(* IEC 61131-3 sources: sigmatek-logger-api/IXON_API/Class/IXON_LoggerAPI_Interface, 1 file *)

(* ---- IXON_LoggerAPI_Interface.st ---- *)
#define SND_DATA_ARRAY_SIZE 1024
#define SND_ARRAY_SIZE 20
#define RCV_DATA_ARRAY_SIZE 1024

(*!
<Class
	Name               = "IXON_LoggerAPI_Interface"
	Revision           = "0.0"
	RealtimeTask       = "false"
	CyclicTask         = "true"
	DefCyclictime      = "10 ms"
	BackgroundTask     = "false"
	Sigmatek           = "false"
	OSInterface        = "false"
	HighPriority       = "false"
	Automatic          = "false"
	UpdateMode         = "Prescan"
	SharedCommandTable = "true"
	Objectsize         = "(810,360)">
	<Channels>
		<Server Name="sIPAddrIXON" Class="String" Visualized="true" Remotely="true" Initialize="true" WriteProtected="false" Retentive="false" Comment="use this channel to access the string functions"/>
		<Server Name="sIPAddrPLC" Class="String" Visualized="true" Remotely="true" Initialize="true" WriteProtected="false" Retentive="false" Comment="use this channel to access the string functions"/>
		<Server Name="sPasswordIXON" Class="String" Visualized="true" Remotely="true" Initialize="true" WriteProtected="false" Retentive="false" Comment="use this channel to access the string functions"/>
		<Server Name="sRcvCnt" Visualized="false" Initialize="false" WriteProtected="true" Retentive="false"/>
		<Server Name="sReconnectDelay" Visualized="true" Remotely="true" Initialize="true" DefValue="10000" WriteProtected="false" Retentive="false"/>
		<Server Name="sSendDelay" Visualized="true" Remotely="true" Initialize="true" DefValue="200" WriteProtected="false" Retentive="false"/>
		<Server Name="sSndCnt" Visualized="false" Initialize="false" WriteProtected="true" Retentive="false"/>
		<Server Name="sTCPStep" Visualized="true" Remotely="true" Initialize="false" WriteProtected="false" Retentive="false"/>
		<Client Name="_StdLib" Required="false" Internal="false"/>
		<Client Name="ST_IPAddrIXON" Required="true" Internal="true"/>
		<Client Name="ST_IPAddrPLC" Required="true" Internal="true"/>
		<Client Name="ST_PasswordIXON" Required="true" Internal="true"/>
	</Channels>
	<Separators>
		<Servers>
			<SepChn Position="0"/>
			<SepChn Position="6"/>
		</Servers>
	</Separators>
	<Network Name="IXON_LoggerAPI_Interface">
		<!-- List of Components in this network -->
		<Components>
			<Object
				Name       = "_base"
				Class      = "_TCPIPClientInterface"
				Position   = "(218,120)"
				Visualized = "false">
				<Channels>
					<Server Name="ClassSvr"/>
					<Server Name="ErrorCode"/>
					<Server Name="ErrorGroup"/>
					<Server Name="ErrorState"/>
					<Server Name="State"/>
					<Client Name="_TCPIPClient"/>
				</Channels>
			</Object>
			<Object
				Name       = "ST_IPAddrIXON"
				Class      = "String"
				Position   = "(210,510)"
				Visualized = "true"
				Remotely   = "true">
				<Channels>
					<Server Name="Data"/>
					<Client Name="SingleRealloc" Value="1"/>
				</Channels>
			</Object>
			<Object
				Name       = "ST_IPAddrPLC"
				Class      = "String"
				Position   = "(210,660)"
				Visualized = "true"
				Remotely   = "true">
				<Channels>
					<Server Name="Data"/>
					<Client Name="SingleRealloc" Value="1"/>
				</Channels>
			</Object>
			<Object
				Name       = "ST_PasswordIXON"
				Class      = "String"
				Position   = "(210,810)"
				Visualized = "true"
				Remotely   = "true">
				<Channels>
					<Server Name="Data"/>
					<Client Name="SingleRealloc" Value="1"/>
				</Channels>
			</Object>
		</Components>
		<Comments>
		</Comments>
		<!-- List of Connections in this network -->
		<Connections>
			<Connection Source="this.ClassSvr" Destination="_base.ClassSvr" Vertices="(1096,210),(924,210),"/>
			<Connection Source="this.State" Destination="_base.State" Vertices="(1096,270),(924,270),"/>
			<Connection Source="this.ErrorState" Destination="_base.ErrorState" Vertices="(1096,330),(924,330),"/>
			<Connection Source="this.ErrorGroup" Destination="_base.ErrorGroup" Vertices="(1096,390),(924,390),"/>
			<Connection Source="this.ErrorCode" Destination="_base.ErrorCode" Vertices="(1096,450),(924,450),"/>
			<Connection Source="_base._TCPIPClient" Destination="this._TCPIPClient" Vertices="(218,210),(38,210),"/>
			<Connection Source="this.ST_IPAddrIXON" Destination="ST_IPAddrIXON.Data"/>
			<Connection Source="this.sIPAddrIXON" Destination="ST_IPAddrIXON.Data" Vertices="(1096,510),(586,600),"/>
			<Connection Source="this.ST_PasswordIXON" Destination="ST_PasswordIXON.Data"/>
			<Connection Source="this.sPasswordIXON" Destination="ST_PasswordIXON.Data" Vertices="(1096,630),(586,900),"/>
			<Connection Source="this.ST_IPAddrPLC" Destination="ST_IPAddrPLC.Data"/>
			<Connection Source="this.sIPAddrPLC" Destination="ST_IPAddrPLC.Data" Vertices="(1096,570),(586,750),"/>
		</Connections>
		<!-- Headerfiles -->
		<Options>
		</Options>
	</Network>
</Class>
*)
#pragma using _TCPIPClientInterface

IXON_LoggerAPI_Interface : CLASS
: _TCPIPClientInterface
	TYPE
	  teUSER_TCP_STEPS :  //! <Type Public="true" Name="teUSER_TCP_STEPS"/>
	  (
	    UTS_Idle,
	    UTS_Connect,
	    UTS_CheckConnect,
	    UTS_ConnectIXON,
	    UTS_WaitConnectIXON,
	    UTS_WaitData,
	    UTS_SendData,
	    UTS_WaitSendData,
	    UTS_Disconnect,
	    UTS_Error
	  )$UDINT;
	END_TYPE
  //Servers:
	sIPAddrIXON 	: SvrChCmd_UDINT;
	sIPAddrPLC 	: SvrChCmd_UDINT;
	sPasswordIXON 	: SvrChCmd_UDINT;
	sSendDelay 	: SvrCh_UDINT;
	sReconnectDelay 	: SvrCh_UDINT;
	sTCPStep 	: SvrCh_teUSER_TCP_STEPS_PTofCls_IXON_LoggerAPI_Interface;
	sSndCnt 	: SvrCh_DINT;
	sRcvCnt 	: SvrCh_DINT;
  //Clients:
	_StdLib 	: CltChCmd__StdLib;
	ST_IPAddrIXON 	: CltChCmd_String;
	ST_PasswordIXON 	: CltChCmd_String;
	ST_IPAddrPLC 	: CltChCmd_String;
  //Variables:
		vSendData : ARRAY [0..SND_ARRAY_SIZE-1, 0..SND_DATA_ARRAY_SIZE-1] OF CHAR;

		vSendDataIndex 	: DINT;
		vRcvData : ARRAY [0..RCV_DATA_ARRAY_SIZE-1] OF CHAR;

		vRcvNewData 	: DINT;
		vLength 	: UDINT;
		vLocIPAddress : ARRAY [0..15] OF CHAR;

		vIsConnected 	: BOOL;
		vTcpTimeOut 	: UDINT;
		vCheckConnectionIXON 	: UDINT;
		vTimeMark 	: UDINT;
		VTimeMark2 	: UDINT;
		vIntError 	: DINT;
		vConnectData : ARRAY [0..100] OF CHAR;

		vSendRepeat 	: DINT;
  //Functions:

	FUNCTION VIRTUAL GLOBAL Init;

	FUNCTION VIRTUAL GLOBAL CyWork
		VAR_INPUT
			EAX 	: UDINT;
		END_VAR
		VAR_OUTPUT
			state (EAX) 	: UDINT;
		END_VAR;
				//! <Function Comment="This Method is called if Data is received (Overwrite it)&#13;&#10;For receiving a spezial amount of Data you have to use the &#13;&#10;DataHandling Methode." Name="Response"/>
	FUNCTION VIRTUAL GLOBAL Response
		VAR_INPUT
			pData 	: ^void;			//! <Variable Comment="Pointer to Data" Name="Response.pData"/>
			udsize 	: UDINT;			//! <Variable Comment="Size of Data" Name="Response.udsize"/>
		END_VAR;

	FUNCTION GLOBAL AddStringToBuffer
		VAR_INPUT
			pData 	: ^void;
			udLen 	: UDINT;
		END_VAR;

	FUNCTION VIRTUAL GLOBAL sIPAddrIXON::Read
		VAR_OUTPUT
			output (EAX) 	: UDINT;
		END_VAR;

	FUNCTION VIRTUAL GLOBAL sIPAddrIXON::Write
		VAR_INPUT
			input (EAX) 	: UDINT;
		END_VAR
		VAR_OUTPUT
			result (EAX) 	: UDINT;
		END_VAR;

	FUNCTION VIRTUAL GLOBAL sIPAddrPLC::Read
		VAR_OUTPUT
			output (EAX) 	: UDINT;
		END_VAR;

	FUNCTION VIRTUAL GLOBAL sIPAddrPLC::Write
		VAR_INPUT
			input (EAX) 	: UDINT;
		END_VAR
		VAR_OUTPUT
			result (EAX) 	: UDINT;
		END_VAR;

	FUNCTION VIRTUAL GLOBAL sPasswordIXON::Read
		VAR_OUTPUT
			output (EAX) 	: UDINT;
		END_VAR;

	FUNCTION VIRTUAL GLOBAL sPasswordIXON::Write
		VAR_INPUT
			input (EAX) 	: UDINT;
		END_VAR
		VAR_OUTPUT
			result (EAX) 	: UDINT;
		END_VAR;
  //Tables:
	FUNCTION @STD
		VAR_OUTPUT
			ret_code	: CONFSTATES;
		END_VAR;
	FUNCTION GLOBAL TAB @CT_;
END_CLASS;

#pragma using String
#pragma usingLtd _StdLib

FUNCTION VIRTUAL GLOBAL IXON_LoggerAPI_Interface::Init
  VAR
  	index : UDINT;
  END_VAR

  if _FirstScan then
    vTcpTimeOut := 2000 ms;
    vCheckConnectionIXON := 10000 ms;
    vTimeMark := ops.tAbsolute := 10000 ms;
  end_if;
END_FUNCTION

FUNCTION VIRTUAL GLOBAL IXON_LoggerAPI_Interface::CyWork
	VAR_INPUT
		EAX 	: UDINT;
	END_VAR
	VAR_OUTPUT
		state (EAX) 	: UDINT;
	END_VAR
  VAR
  	retCode : DINT;
    index : UDINT;
    length : UDINT;
    i : INT;
  END_VAR

  // ==========================================================================
  case sTCPStep of

    // --------------------------------------------------------------
    UTS_Idle:
      if (ops.tAbsolute - vTimeMark) > 1000 ms then
        sTCPStep := UTS_Connect;
      end_if;

    // --------------------------------------------------------------
    UTS_Connect:

      vLength := ST_IPAddrIXON.GetLength();

      if vLength > sizeof(vLocIPAddress) then
        vTimeMark := ops.tAbsolute;
        vIntError := -1; // IP address too long.
        sTCPStep := UTS_Error;
        return;
      end_if;

      ST_IPAddrIXON.GetDataAt(pData:=#vLocIPAddress[0],
                                 udSize:=vLength,
                                 udAt:=0);

      vLocIPAddress[vLength]:=0;

      retCode := AddConnection(pIPAddress:=#vLocIPAddress[0],
                               udTimeout:= 0);

      if retCode > 0 then
        vTimeMark := ops.tAbsolute;
        sTCPStep := UTS_CheckConnect;
      else
        vTimeMark := ops.tAbsolute;
        vIntError := -2; // Connection could not be established.
        sTCPStep := UTS_Error;
        return;
      end_if;

    // --------------------------------------------------------------
    UTS_CheckConnect:

      if vRcvNewData = 1 then
        vRcvNewData := 0;
        if _memcmp(ptr1:=#vRcvData[0], ptr2:="HELO", cntr:=4) = 0 then
          sTCPStep := UTS_ConnectIXON;
        end_if;
      end_if;
      if (ops.tAbsolute - vTimeMark) > vTcpTimeOut  then
        sTCPStep := UTS_Disconnect;
      end_if;

    // --------------------------------------------------------------
    UTS_ConnectIXON:

      _strcpy(dest:=#vConnectData[0], src:="DEVC ");
      length := ST_IPAddrPLC.GetLength();
      ST_IPAddrPLC.GetDataAt(pData:=#vConnectData[5], udSize:=length, udAt:=0);
      index := 5 + length;
      _strcat(dest:=#vConnectData[index], src:=" ");
      length := ST_PasswordIXON.GetLength();
      index := index + 1;
      ST_PasswordIXON.GetDataAt(pData:=#vConnectData[index], udSize:=length, udAt:=0);
      index := index + length;
      vConnectData[index] := 16#0a;
      vConnectData[index + 1] := 0;

      retCode := SendData(pData:=#vConnectData[0],
                          udSize:= index + 1,
                          bDirect:=TRUE);

      if retCode = 0 then
        vTimeMark := ops.tAbsolute;
        sTCPStep := UTS_WaitConnectIXON;
      else
        vTimeMark := ops.tAbsolute;
        vIntError := -11; // Error connecting IXON
        sTCPStep := UTS_Error;
        return;
      end_if;

    // --------------------------------------------------------------
    UTS_WaitConnectIXON:

      if vRcvNewData = 1 then
        vRcvNewData := 0;
        if _memcmp(ptr1:=#vRcvData[0], ptr2:="DEVC OK", cntr:=7) = 0 then
          vTimeMark := ops.tAbsolute;
          sTCPStep := UTS_WaitData;
        end_if;
      end_if;
      if (ops.tAbsolute - vTimeMark) > vTcpTimeOut  then
        vIntError := -12; // Error connecting IXON response
        sTCPStep := UTS_Error;
      end_if;

    // --------------------------------------------------------------
    UTS_WaitData:

      vIsConnected := IsConnected();

      if vIsConnected = FALSE then
        sTCPStep := UTS_Disconnect;
      elsif _strlen(src:=#vSendData[0][0]) > 0 & (ops.tAbsolute - VTimeMark2) > sSendDelay then
        sTCPStep := UTS_SendData;
      elsif (ops.tAbsolute - vTimeMark) > vCheckConnectionIXON  then
        sTCPStep := UTS_ConnectIXON;
      end_if;

    // --------------------------------------------------------------
    UTS_SendData:

      retCode := SendData(pData:=#vSendData[0][0],
                          udSize:= _strlen(src:=#vSendData[0][0]),
                          bDirect:=TRUE);

      if retCode = 0 then
        for i := 0 to SND_ARRAY_SIZE - 2 do
          vSendData[i] := vSendData[i + 1];
        end_for;
        _strcpy(dest:=#vSendData[SND_ARRAY_SIZE - 1][0], src:="");
        vSendDataIndex -= 1;

        sSndCnt += 1;
        vTimeMark := ops.tAbsolute;
        vTimeMark2 := ops.tAbsolute;
        vSendRepeat := 0;
        sTCPStep := UTS_WaitData; //UTS_WaitSendData;
      else
        vTimeMark := ops.tAbsolute;
        vIntError := -3; // Error sending data
        sTCPStep := UTS_Error;
        return;
      end_if;

    // --------------------------------------------------------------
    UTS_WaitSendData:

      if (ops.tAbsolute - vTimeMark) > vTcpTimeOut  then
        sTCPStep := UTS_Disconnect;
      end_if;

    // --------------------------------------------------------------
    UTS_Disconnect:

      retCode := DelConnection();

      if retCode  = TCP_CLT_NO_ERROR then
        vTimeMark := ops.tAbsolute;
        sTCPStep := UTS_Idle;
      else
        vTimeMark := ops.tAbsolute;
        vIntError := -4; // Error while closing the connection.
        sTCPStep := UTS_Error;
        return;
      end_if;

    // --------------------------------------------------------------
    UTS_Error:
      if vIntError = -2 & (ops.tAbsolute - vTimeMark) > sReconnectDelay then //Connect error
        sTCPStep := UTS_Connect;
      elsif vIntError = -3 then //Send error, retry 3 times, then stay in error
        vSendRepeat := vSendRepeat + 1;
        if vSendRepeat < 3 then
          sTCPStep := UTS_SendData;
        end_if;
      elsif vIntError <= -11 then //IXON Connect error
        sTCPStep := UTS_DISConnect;
      end_if;

  end_case;
  // ==========================================================================

	state := READY;

END_FUNCTION

FUNCTION VIRTUAL GLOBAL IXON_LoggerAPI_Interface::Response
	VAR_INPUT
		pData 	: ^void;
		udsize 	: UDINT;
	END_VAR
  VAR
  	pDest : ^void;
  END_VAR

  sRcvCnt += 1;

  pDest:= _StdLib.MemSet(dest:=#vRcvData[0],
                         value:=0,
                         size:=sizeof(vRcvData));

  if pDest <> #vRcvData[0] then
    vIntError := -5;
    sTCPStep := UTS_Error;
    return;
  end_if;

  if udsize > sizeof(vRcvData) then
    udsize := sizeof(vRcvData);
  end_if;

  pDest := _StdLib.MemCpy(dest:=#vRcvData[0],
                          source:=pData,
                          size:=udsize);

  if pDest <> #vRcvData[0] then
    vIntError := -6;
    sTCPStep := UTS_Error;
    return;
  end_if;

  vRcvNewData := 1;

END_FUNCTION

FUNCTION VIRTUAL GLOBAL IXON_LoggerAPI_Interface::sIPAddrIXON::Read
	VAR_OUTPUT
		output (EAX) 	: UDINT;
	END_VAR

	sIPAddrIXON := ST_IPAddrIXON.Data.Read();
	output := sIPAddrIXON;

END_FUNCTION

FUNCTION VIRTUAL GLOBAL IXON_LoggerAPI_Interface::sIPAddrIXON::Write
	VAR_INPUT
		input (EAX) 	: UDINT;
	END_VAR
	VAR_OUTPUT
		result (EAX) 	: UDINT;
	END_VAR

	sIPAddrIXON := input;
	result := (ST_IPAddrIXON.Data.Write(sIPAddrIXON))$UDINT;

END_FUNCTION

FUNCTION VIRTUAL GLOBAL IXON_LoggerAPI_Interface::sPasswordIXON::Read
	VAR_OUTPUT
		output (EAX) 	: UDINT;
	END_VAR

	sPasswordIXON := ST_PasswordIXON.Data.Read();
	output := sPasswordIXON;

END_FUNCTION

FUNCTION VIRTUAL GLOBAL IXON_LoggerAPI_Interface::sPasswordIXON::Write
	VAR_INPUT
		input (EAX) 	: UDINT;
	END_VAR
	VAR_OUTPUT
		result (EAX) 	: UDINT;
	END_VAR

	sPasswordIXON := input;
	result := (ST_PasswordIXON.Data.Write(sPasswordIXON))$UDINT;

END_FUNCTION

FUNCTION VIRTUAL GLOBAL IXON_LoggerAPI_Interface::sIPAddrPLC::Read
	VAR_OUTPUT
		output (EAX) 	: UDINT;
	END_VAR

	sIPAddrPLC := ST_IPAddrPLC.Data.Read();
	output := sIPAddrPLC;

END_FUNCTION

FUNCTION VIRTUAL GLOBAL IXON_LoggerAPI_Interface::sIPAddrPLC::Write
	VAR_INPUT
		input (EAX) 	: UDINT;
	END_VAR
	VAR_OUTPUT
		result (EAX) 	: UDINT;
	END_VAR

	sIPAddrPLC := input;
	result := (ST_IPAddrPLC.Data.Write(sIPAddrPLC))$UDINT;

END_FUNCTION

FUNCTION GLOBAL IXON_LoggerAPI_Interface::AddStringToBuffer
	VAR_INPUT
		pData 	: ^void;
		udLen 	: UDINT;
	END_VAR
  VAR
  	i : DINT;
  END_VAR

  if vSendDataIndex <= SND_ARRAY_SIZE - 1 then
    _StdLib.memcpy(dest:=#vSendData[vSendDataIndex][0], source:=pData, size:=udLen);
    vSendDataIndex += 1;
  else
    //Move buffer 1 position and add string at end of buffer
    for i := 0 to SND_ARRAY_SIZE - 2 do
      vSendData[i] := vSendData[i + 1];
    end_for;
    _StdLib.memcpy(dest:=#vSendData[SND_ARRAY_SIZE - 1][0], source:=pData, size:=udLen);
  end_if;
END_FUNCTION
